{attribute 'GeneratedUsingTerminal: EK1122-0000-0018'}
{attribute addProperty BoxType "EK1122-0000-0018"}
{attribute addProperty Id "Beckhoff_EP4xxxsub_EK1100EK1100_1FC0878B2A_0001_EP4174_0002_0016EP4174_D2A7C9B719A_0002_EP4174_0002_0017EP4174_D2A7C9B719A_0003_EP4174_0002_0018EP4174_D2A7C9B719A_0004_EP4174_0002_0019EP4174_D2A7C9B719A_0005_EP4314_1002_0016EP4314_1D6CF30B38A_0006_EP4374_0002_0016EP4374_4CDC402D36A_0007_EP4374_0002_0017EP4374_6231FEFD36A_0008_EP4374_0002_0018EP4374_6231FEFD36A_0009_EP4374_0002_0019EP4374_6231FEFD36A_0010_EP4378_1022_0017EP4378_DC3B21DF76"}
{attribute addProperty CRC "509565897"}
{attribute addProperty Size "336"}
TYPE Beckhoff_EP4xxxEK1122_1E5F5BC9 EXTENDS EK1122_1FC0878B :
STRUCT
	{attribute addProperty Name "Beckhoff_EP4xxxsub_EK1100"}
	{attribute addProperty PreviousPort "Beckhoff EP4xxxEK1122 : D"}
	Beckhoff_EP4xxxsub_EK1100 : EK1100_1FC0878B;
	{attribute addProperty Name "A_0001_EP4174_0002_0016"}
	{attribute addProperty PreviousPort "Beckhoff EP4xxxsub EK1100 : C"}
	A_0001_EP4174_0002_0016 : EP4174_D2A7C9B7;
	{attribute addProperty Name "A_0002_EP4174_0002_0017"}
	{attribute addProperty PreviousPort "A_0001(EP4174-0002-0016) : B"}
	A_0002_EP4174_0002_0017 : EP4174_D2A7C9B7;
	{attribute addProperty Name "A_0003_EP4174_0002_0018"}
	{attribute addProperty PreviousPort "A_0002(EP4174-0002-0017) : B"}
	A_0003_EP4174_0002_0018 : EP4174_D2A7C9B7;
	{attribute addProperty Name "A_0004_EP4174_0002_0019"}
	{attribute addProperty PreviousPort "A_0003(EP4174-0002-0018) : B"}
	A_0004_EP4174_0002_0019 : EP4174_D2A7C9B7;
	{attribute addProperty Name "A_0005_EP4314_1002_0016"}
	{attribute addProperty PreviousPort "A_0004(EP4174-0002-0019) : B"}
	A_0005_EP4314_1002_0016 : EP4314_1D6CF30B;
	{attribute addProperty Name "A_0006_EP4374_0002_0016"}
	{attribute addProperty PreviousPort "A_0005(EP4314-1002-0016) : B"}
	A_0006_EP4374_0002_0016 : EP4374_4CDC402D;
	{attribute addProperty Name "A_0007_EP4374_0002_0017"}
	{attribute addProperty PreviousPort "A_0006(EP4374-0002-0016) : B"}
	A_0007_EP4374_0002_0017 : EP4374_6231FEFD;
	{attribute addProperty Name "A_0008_EP4374_0002_0018"}
	{attribute addProperty PreviousPort "A_0007(EP4374-0002-0017) : B"}
	A_0008_EP4374_0002_0018 : EP4374_6231FEFD;
	{attribute addProperty Name "A_0009_EP4374_0002_0019"}
	{attribute addProperty PreviousPort "A_0008(EP4374-0002-0018) : B"}
	A_0009_EP4374_0002_0019 : EP4374_6231FEFD;
	{attribute addProperty Name "A_0010_EP4378_1022_0017"}
	{attribute addProperty PreviousPort "A_0009(EP4374-0002-0019) : B"}
	A_0010_EP4378_1022_0017 : EP4378_DC3B21DF;
END_STRUCT
END_TYPE

(* stored: Version 1.2.0.0, ProductVersion 3.1.4024.9
   DUT Beckhoff_EP4xxxEK1122_1E5F5BC9: Id {4e0f44f4-3eef-40f0-a32f-4b23bbe136bd} *)
